// TIA Portal V20 export
DATA_BLOCK "EQUIPMENT_DATA_GLOBAL_DB"   // DB200
{ S7_Optimized_Access := 'TRUE' }
// stored: AutoNumber false, MemoryReserve 100
   VAR RETAIN
      EmptyStepHistory { S7_SetPoint := 'True'} : Array[0.."EQUIPMENTDATA_STEPHISTORYLENGTH"] of "GRAPH_STEP_HISTORY_UDT";
   END_VAR
   VAR
      Dummy_IF_COND { ExternalAccessible := 'False'; ExternalVisible := 'False'; ExternalWritable := 'False'; S7_SetPoint := 'True'} : "COND_PD_UDT";
   END_VAR
BEGIN
END_DATA_BLOCK
